// Mitsubishi GX Works2 project: 20240117_AI机程序新增旋钮开关   PLC: FX3S

PROGRAM MAIN
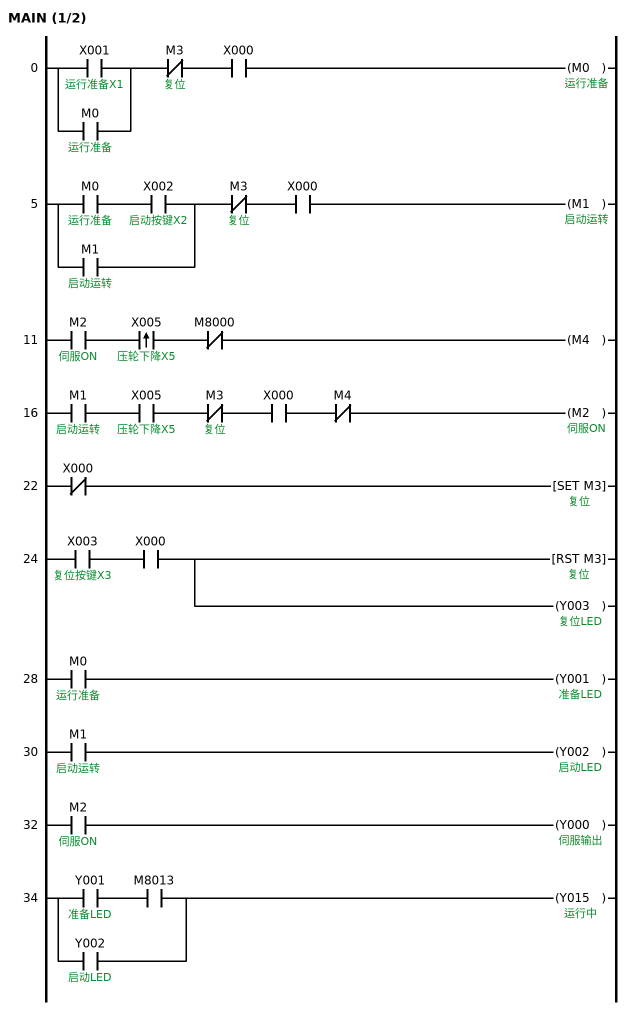
0     LD      X001  ; 运行准备X1
      OR      M0  ; 运行准备
      ANI     M3  ; 复位
      AND     X000
      OUT     M0  ; 运行准备
5     LD      M0  ; 运行准备
      AND     X002  ; 启动按键X2
      OR      M1  ; 启动运转
      ANI     M3  ; 复位
      AND     X000
      OUT     M1  ; 启动运转
11    LD      M2  ; 伺服ON
      ANDP    X005  ; 压轮下降X5
      ANI     M8000
      OUT     M4
16    LD      M1  ; 启动运转
      AND     X005  ; 压轮下降X5
      ANI     M3  ; 复位
      AND     X000
      ANI     M4
      OUT     M2  ; 伺服ON
22    LDI     X000
      SET     M3  ; 复位
24    LD      X003  ; 复位按键X3
      AND     X000
      RST     M3  ; 复位
      OUT     Y003  ; 复位LED
28    LD      M0  ; 运行准备
      OUT     Y001  ; 准备LED
30    LD      M1  ; 启动运转
      OUT     Y002  ; 启动LED
32    LD      M2  ; 伺服ON
      OUT     Y000  ; 伺服输出
34    LD      Y001  ; 准备LED
      AND     M8013
      OR      Y002  ; 启动LED
      OUT     Y015  ; 运行中
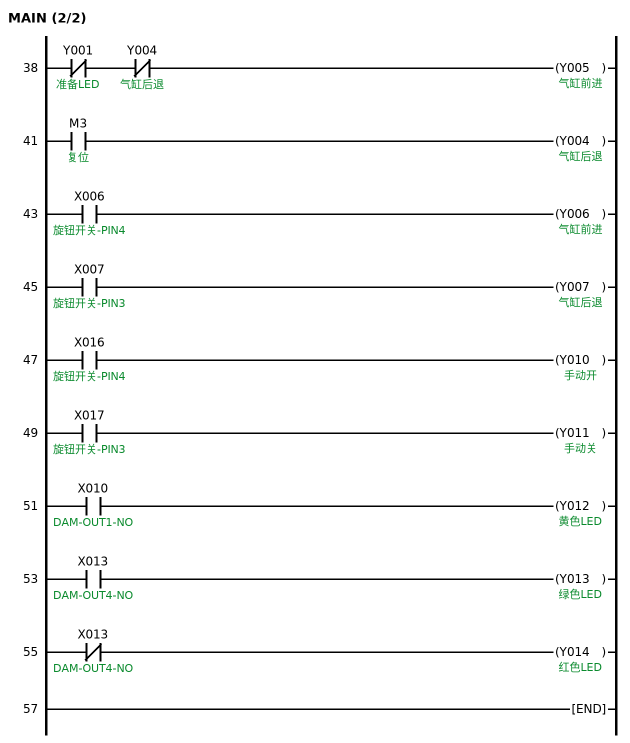
38    LDI     Y001  ; 准备LED
      ANI     Y004  ; 气缸后退
      OUT     Y005  ; 气缸前进
41    LD      M3  ; 复位
      OUT     Y004  ; 气缸后退
43    LD      X006  ; 旋钮开关-PIN4
      OUT     Y006  ; 气缸前进
45    LD      X007  ; 旋钮开关-PIN3
      OUT     Y007  ; 气缸后退
47    LD      X016  ; 旋钮开关-PIN4
      OUT     Y010  ; 手动开
49    LD      X017  ; 旋钮开关-PIN3
      OUT     Y011  ; 手动关
51    LD      X010  ; DAM-OUT1-NO
      OUT     Y012  ; 黄色LED
53    LD      X013  ; DAM-OUT4-NO
      OUT     Y013  ; 绿色LED
55    LDI     X013  ; DAM-OUT4-NO
      OUT     Y014  ; 红色LED
57    END
END_PROGRAM

// device comments not shown above
X011  ; DAM-OUT2-NO
X012  ; DAM-OUT3-NO
X014  ; DAM-OUT5-NO
X015  ; DAM-OUT6-NO
